FUNCTION HYST_3 (* Hystereses function *)
  (* Standard: 61499-1 *)
  (* Version 1.0, 2025-12-21, franz *)
  PACKAGE OSCAT::Basic::POUs::Engineering::Control;
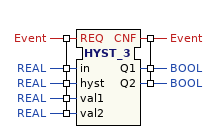
  EVENT_INPUT
    REQ WITH in, hyst, val1, val2;
  END_EVENT
  EVENT_OUTPUT
    CNF WITH Q1, Q2;
  END_EVENT
  VAR_INPUT
    in : REAL;
    hyst : REAL;
    val1 : REAL;
    val2 : REAL;
  END_VAR
  VAR_OUTPUT
    Q1 : BOOL;
    Q2 : BOOL;
  END_VAR
  BODY IN ST:
PACKAGE OSCAT::Basic::POUs::Engineering::Control;

(* Hystereses function *)
FUNCTION HYST_3
VAR_INPUT
	in : REAL;
	hyst : REAL;
	val1 : REAL;
	val2 : REAL;
END_VAR
VAR_OUTPUT
	Q1 : BOOL;
	Q2 : BOOL;
END_VAR
VAR
	X : REAL;
END_VAR

(*
 * version 1.2	5 jan 2008 programmer 	oscat tested BY	oscat
 * *
 * this is a double hysteresis function. Out1 follows a hysteresis function defined by val1and hyst,
 * while out 2 follows val2 and hyst.
 * if the input signal is between the two hysteresis switches (val1 and val2) then non of the
 * outputs is active.
 *)
X := hyst * 0.5;
IF in < val1 - X THEN
	Q1 := TRUE;
ELSIF in > val1 + X THEN
	Q1 := FALSE;
END_IF;
IF in < val2 - X THEN
	Q2 := FALSE;
ELSIF in > val2 + X THEN
	Q2 := TRUE;
END_IF;

END_FUNCTION

(* revision history hm	22. jan 2007	rev 1.0 original version
 * *
 * hm	27. dec 2007	rev 1.1 changed code for better performance
 * *
 * hm	5. jan 2008	rev 1.2 further performance iprovements *)
  END_BODY
END_FUNCTION
